{attribute addProperty BoxType "EK1100-0000-0018"}
{attribute addProperty Id "InfoDataInfoData_FC4995DF11214"}
{attribute addProperty CRC "3958522194"}
{attribute addProperty SizeInBites "112"}
{attribute addProperty SizeInBytes "14"}
TYPE EK1100_EBF24152 :
STRUCT
	{attribute addProperty Name "InfoData"}
	InfoData : InfoData_FC4995DF;
END_STRUCT
END_TYPE

(* stored: Version 1.2.0.0, ProductVersion 3.1.4024.9
   DUT EK1100_EBF24152: Id {258a4e8e-01f3-0b67-21f0-e5b9843d9077} *)
